{attribute 'qualified_only'}
VAR_GLOBAL
//Atrium
	strEnOceanSwitch_Gang_3_109_PladeA				: Tc2_EnOcean.STR_EnOceanSwitch;
	strEnOceanSwitch_AtriumNiveau_PladeB				: Tc2_EnOcean.STR_EnOceanSwitch;
	strEnOceanSwitch_AtriumNiveau_Service				: Tc2_EnOcean.STR_EnOceanSwitch;
	

//Gange
	strEnOceanSwitch_Gang_7_301				: Tc2_EnOcean.STR_EnOceanSwitch;

	//Rum
	strEnOceanSwitch_Rum_2_341_Indgang		: Tc2_EnOcean.STR_EnOceanSwitch;
	strEnOceanSwitch_Rum_2_341_Ekstra		: Tc2_EnOcean.STR_EnOceanSwitch;
    strEnOceanSwitch_Rum_2_345      : Tc2_EnOcean.STR_EnOceanSwitch;
	strEnOceanSwitch_Rum_2_345_Ekstra		: Tc2_EnOcean.STR_EnOceanSwitch;
	strEnOceanSwitch_Rum_2_349				: Tc2_EnOcean.STR_EnOceanSwitch;
	
	
END_VAR

(* stored: Version 1.1.0.1
   GVL GVL_EnOcean: Id {bec68ff9-8f1d-4ce1-b8b9-84de691aacc9} *)
